DATA_BLOCK "群控调度_DB"
{ S7_Optimized_Access := 'TRUE' }
VERSION : 0.1
NON_RETAIN
"群控调度"

BEGIN

END_DATA_BLOCK

